// TIA Portal V20 export
DATA_BLOCK "BK14"   // DB292
// stored: MemoryReserve 100
   VAR
      "X10-1.FIX CATHODE FRONT BACKWARD" : Bool := FALSE;
      "X11-1.STACK TABLE OUT REAR Z-AXIS LIMIT SENSOR(-)" : Bool := TRUE;
      "X12-1.FIX CATHODE REAR BACKWARD" : Bool := FALSE;
      "X13-1.STACK TABLE OUT REAR Z-AXIS LIMIT SENSOR(+)" : Bool := TRUE;
      "X14-1.FIX CATHODE DETECT SENSOR" : Bool := FALSE;
      "X15-1.SPARE" : Bool := FALSE;
      "X16-1.SPARE" : Bool := FALSE;
      "X17-1.SPARE" : Bool := FALSE;
      "X10-2.FIX CATHODE FRONT FORWARD" : Bool := TRUE;
      "X11-2.STACK TABLE OUT REAR Z-AXIS HOME SENSOR" : Bool := TRUE;
      "X12-2.FIX CATHODE REAR FORWARD" : Bool := TRUE;
      "X13-2.SPARE" : Bool := FALSE;
      "X14-2.SPARE" : Bool := FALSE;
      "X15-2.SPARE" : Bool := FALSE;
      "X16-2.SPARE" : Bool := FALSE;
      "X17-2.SPARE" : Bool := FALSE;
   END_VAR
BEGIN
END_DATA_BLOCK
